SUBAPPLICATION Uebung_030 (* LED_PWM Blinkende LED *)
  (* Standard: 61499-2 *)
  (* Version 1.0, 2023-10-23, franz *)
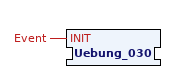
  EVENT_INPUT
    INIT;
  END_EVENT
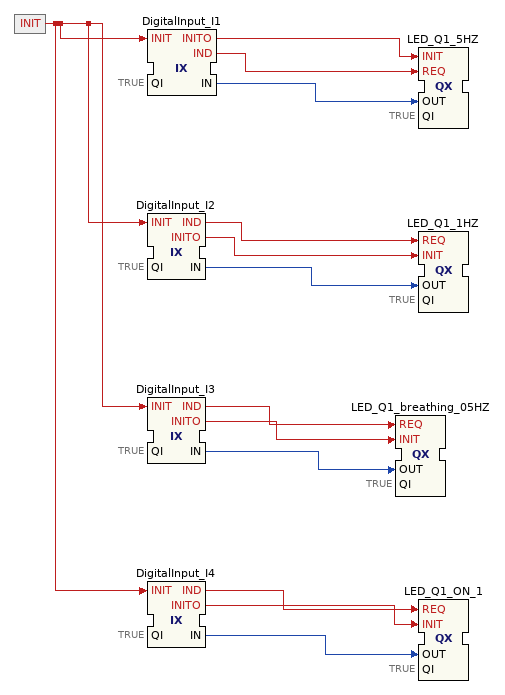
  FBS
    LED_Q1_5HZ : QX(QI := TRUE);
    DigitalInput_I1 : IX(QI := TRUE);
    LED_Q1_1HZ : QX(QI := TRUE);
    DigitalInput_I2 : IX(QI := TRUE);
    LED_Q1_breathing_05HZ : QX(QI := TRUE);
    DigitalInput_I3 : IX(QI := TRUE);
    DigitalInput_I4 : IX(QI := TRUE);
    LED_Q1_ON_1 : QX(QI := TRUE);
  END_FBS
  EVENT_CONNECTIONS
    INIT TO DigitalInput_I1.INIT;
    DigitalInput_I1.INITO TO LED_Q1_5HZ.INIT;
    DigitalInput_I1.IND TO LED_Q1_5HZ.REQ;
    DigitalInput_I2.IND TO LED_Q1_1HZ.REQ;
    INIT TO DigitalInput_I2.INIT;
    DigitalInput_I2.INITO TO LED_Q1_1HZ.INIT;
    INIT TO DigitalInput_I3.INIT;
    DigitalInput_I3.IND TO LED_Q1_breathing_05HZ.REQ;
    DigitalInput_I3.INITO TO LED_Q1_breathing_05HZ.INIT;
    DigitalInput_I4.IND TO LED_Q1_ON_1.REQ;
    DigitalInput_I4.INITO TO LED_Q1_ON_1.INIT;
    INIT TO DigitalInput_I4.INIT;
  END_CONNECTIONS
  DATA_CONNECTIONS
    DigitalInput_I1.IN TO LED_Q1_5HZ.OUT;
    DigitalInput_I2.IN TO LED_Q1_1HZ.OUT;
    DigitalInput_I3.IN TO LED_Q1_breathing_05HZ.OUT;
    DigitalInput_I4.IN TO LED_Q1_ON_1.OUT;
  END_CONNECTIONS
END_SUBAPPLICATION
